(* PLC project faults, TNI-Software ControlBuild 4.00.17 *)
(* stored: creationDateTime 2005-06-20T11:53:06-01:00 *)

FUNCTION_BLOCK cmd_equipment_library.faults
  VAR_INPUT  (* CB.group=Orders CB.kind=inputVars *)
    workCmd : BOOL := false;  (* CB.mnemonicPatternPropertyName=<SY>_CMDFW_<NU> CB.libelle=Work command to the valve *)
    restCmd : BOOL := false;  (* CB.mnemonicPatternPropertyName=<SY>_CMDS_<NU> CB.libelle=Rest command to the valve *)
  END_VAR
  VAR_INPUT  (* CB.group=Sensors CB.kind=inputVars *)
    outletSensor : BOOL := false;  (* CB.libelle=Outlet sensor *)
    inletSensor : BOOL := false;  (* CB.libelle=Inlet sensor *)
  END_VAR
  VAR_INPUT  (* CB.kind=inputVars *)
    acknowledgePB : BOOL := false;  (* CB.mnemonicPatternPropertyName=<SY>PBACK<NU> CB.libelle=Acknowledgement pushbutton *)
  END_VAR
  VAR_OUTPUT  (* CB.kind=outputVars *)
    generalFault : BOOL := false;  (* CB.mnemonicPatternPropertyName=grlFlt<SY><NU> CB.libelle=General fault of the jack *)
  END_VAR
  VAR CONSTANT  (* CB.kind=parameterVars *)
    presetMvt : DINT := 2;  (* CB.mnemonicPatternPropertyName=presetMvt<SY><NU> CB.libelle=in seconds *)
    presetDiscordance : DINT := 200;  (* CB.mnemonicPatternPropertyName=presetDisc<SY><NU> CB.libelle=in milliseconds *)
  END_VAR
  VAR  (* CB.group=Faults CB.kind=overControlVars *)
    discordanceFault : BOOL := false;  (* CB.mnemonicPatternPropertyName=discFlt<SY><NU> CB.libelle=Discordance between sensors *)
    outletSensorFault : BOOL := false;  (* CB.mnemonicPatternPropertyName=outletFlt<SY><NU> CB.libelle=Outlet sensor fault *)
    inletSensorFault : BOOL := false;  (* CB.mnemonicPatternPropertyName=inletFlt<SY><NU> CB.libelle=Inlet sensor fault *)
  END_VAR

(* LD diagram, written out as Structured Text *)
1:
IF acknowledgePB THEN discordanceFault := FALSE; END_IF;
IF acknowledgePB THEN outletSensorFault := FALSE; END_IF;
IF acknowledgePB THEN inletSensorFault := FALSE; END_IF;
IF acknowledgePB THEN generalFault := FALSE; END_IF;
2:
ton_sec_1(IN := workCmd, PT := presetMvt);
IF ton_sec_1.Q AND NOT outletSensor THEN outletSensorFault := TRUE; END_IF;
ton_sec_2(IN := restCmd, PT := presetMvt);
IF ton_sec_2.Q AND NOT inletSensor THEN inletSensorFault := TRUE; END_IF;
3:
ton_ms_3(IN := outletSensor AND inletSensor, PT := presetDiscordance);
IF ton_ms_3.Q THEN discordanceFault := TRUE; END_IF;
4:
IF discordanceFault OR outletSensorFault OR inletSensorFault THEN generalFault := TRUE; END_IF;
END_FUNCTION_BLOCK
